INTERFACE I_LogArgument EXTENDS I_Base

METHOD ToString : T_MaxString
VAR_INPUT
END_VAR
END_METHOD

END_INTERFACE

(* stored: Version 1.1.0.1, ProductVersion 3.1.4026.18
   Itf I_LogArgument: Id {95a4d088-a376-4390-9a94-3d18bd923c60}
   Method ToString: Id {0ce7c76a-4408-45f3-b331-943b4f7839a6} *)
